// TIA Portal V18 export
// export: Created 2026-06-24T03:56:38.2545712Z, ExportSetting WithDefaults, DisplayName Totally Integrated Automation Portal, DisplayVersion V18, DisplayName TIA Portal Openness, DisplayVersion V18, DisplayName TIA Portal Version Control Interface, DisplayVersion V18, DisplayName STEP 7 Professional, DisplayVersion V18, DisplayName STEP 7 Safety, DisplayVersion V18, DisplayName WinCC Professional, DisplayVersion V18
ORGANIZATION_BLOCK "Cyclic interrupt"   // OB30, LAD, CyclicInterrupt
{ S7_Optimized_Access := 'TRUE' }
VERSION : 0.1
// stored: AutoNumber true, IsIECCheckEnabled false, SetENOAutomatically false
   VAR_INPUT
      Initial_Call : Bool;   // Initial call of this OB
      Event_Count : Int;   // Events discarded
   END_VAR
BEGIN

REGION Network 1
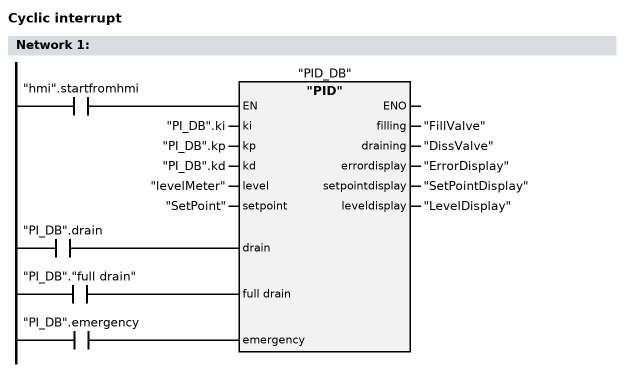
   RUNG wire#powerrail
      Contact( "hmi".startfromhmi )
      "PID_DB"(drain := wire#w1, "full drain" := wire#w2, emergency := wire#w3, ki := "PI_DB".ki, kp := "PI_DB".kp, kd := "PI_DB".kd, level := "levelMeter", setpoint := "SetPoint", filling => "FillValve", draining => "DissValve", errordisplay => "ErrorDisplay", setpointdisplay => "SetPointDisplay", leveldisplay => "LevelDisplay")
   END_RUNG
   RUNG wire#powerrail
      Contact( "PI_DB".drain )
   END_RUNG wire#w1
   RUNG wire#powerrail
      Contact( "PI_DB"."full drain" )
   END_RUNG wire#w2
   RUNG wire#powerrail
      Contact( "PI_DB".emergency )
   END_RUNG wire#w3
   // the same network as SCL:
   IF "hmi".startfromhmi THEN
       "PID_DB"(ki := "PI_DB".ki,   // "PID"
                kp := "PI_DB".kp,
                kd := "PI_DB".kd,
                level := "levelMeter",
                setpoint := "SetPoint",
                drain := "PI_DB".drain,
                "full drain" := "PI_DB"."full drain",
                emergency := "PI_DB".emergency,
                filling => "FillValve",
                draining => "DissValve",
                errordisplay => "ErrorDisplay",
                setpointdisplay => "SetPointDisplay",
                leveldisplay => "LevelDisplay");
   END_IF;
END_REGION

REGION Network 2 (SCL): TO BE SURE THAT KP ON PID WILL BE ALWAYS BIGGER THAN 1
   IF "PI_DB".kp < 1 THEN
       "PI_DB".kp := 1;
   END_IF;
END_REGION
END_ORGANIZATION_BLOCK
